(* Schneider Machine Expert - Basic project DFS, file version 2.5.0.0 *)
(* ProjectInformations: Name=New project *)

HARDWARE
  Cpu 0: TM221CE24R
  EthernetConfiguration: NetworkName=M221, IpAllocationMode=FixedAddress, IpAddress=0.0.0.0, SubnetMask=0.0.0.0
  SerialLineConfiguration: Baud=Baud19200, Parity=ParityEven, DataBits=DataBits8, StopBits=StopBits1, PhysicalMedium=PhysicalMediumRs485, TransmissionMode=TransmissionModeModbusRtu, SlaveId=1, Addressing=SlaveAddressing
  MastTask: UsePeriodScanMode=false, PeriodScan=100
  FastTask: Period=255
  CpuBehavior: StartingMode=StartAsPreviousState, AutoSaveRamOnEeprom=true, WatchdogPeriod=250

SYMBOLS  (address, symbol, comment, settings)
  %M0       SENSOR_JARAK_BIT
  %M1       LEVEL_BIT
  %M2       SM_BIT
  %M3       SB_BIT
  %M4       MOTOR_BIT
  %M5       WADAH_KT_BIT
  %M6       WADAH_KA_BIT
  %M7       MOTOR_TRIG
  %M8       KA_TRIGG
  %M9       KT_TRIG
  %I0.0     SENSOR_JARAK
  %I0.1     LEVEL
  %I0.2     SENSOR_MERAH
  %I0.3     SENSOR_BIRU
  %Q0.0     MOTOR_CONVEYOR
  %Q0.1     WADAH_KT
  %Q0.2     WADAH_KA

POU IO
  (* SectionNumber=0 *)

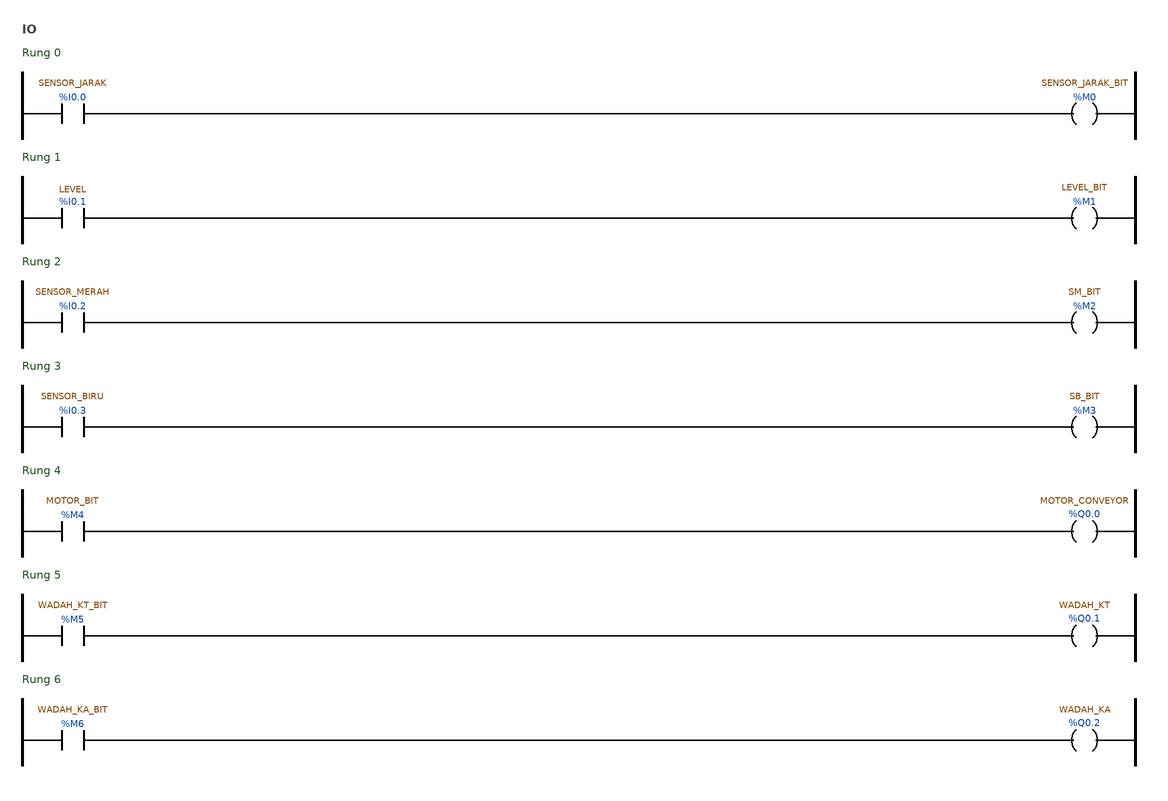

// Rung 0
  LD %I0.0                (* SENSOR_JARAK *)
  ST %M0                  (* SENSOR_JARAK_BIT *)
  // as ST:
  //   SENSOR_JARAK_BIT := SENSOR_JARAK;

// Rung 1
  LD %I0.1                (* LEVEL *)
  ST %M1                  (* LEVEL_BIT *)
  // as ST:
  //   LEVEL_BIT := LEVEL;

// Rung 2
  LD %I0.2                (* SENSOR_MERAH *)
  ST %M2                  (* SM_BIT *)
  // as ST:
  //   SM_BIT := SENSOR_MERAH;

// Rung 3
  LD %I0.3                (* SENSOR_BIRU *)
  ST %M3                  (* SB_BIT *)
  // as ST:
  //   SB_BIT := SENSOR_BIRU;

// Rung 4
  LD %M4                  (* MOTOR_BIT *)
  ST %Q0.0                (* MOTOR_CONVEYOR *)
  // as ST:
  //   MOTOR_CONVEYOR := MOTOR_BIT;

// Rung 5
  LD %M5                  (* WADAH_KT_BIT *)
  ST %Q0.1                (* WADAH_KT *)
  // as ST:
  //   WADAH_KT := WADAH_KT_BIT;

// Rung 6
  LD %M6                  (* WADAH_KA_BIT *)
  ST %Q0.2                (* WADAH_KA *)
  // as ST:
  //   WADAH_KA := WADAH_KA_BIT;

POU CONTROL
  (* SectionNumber=0 *)

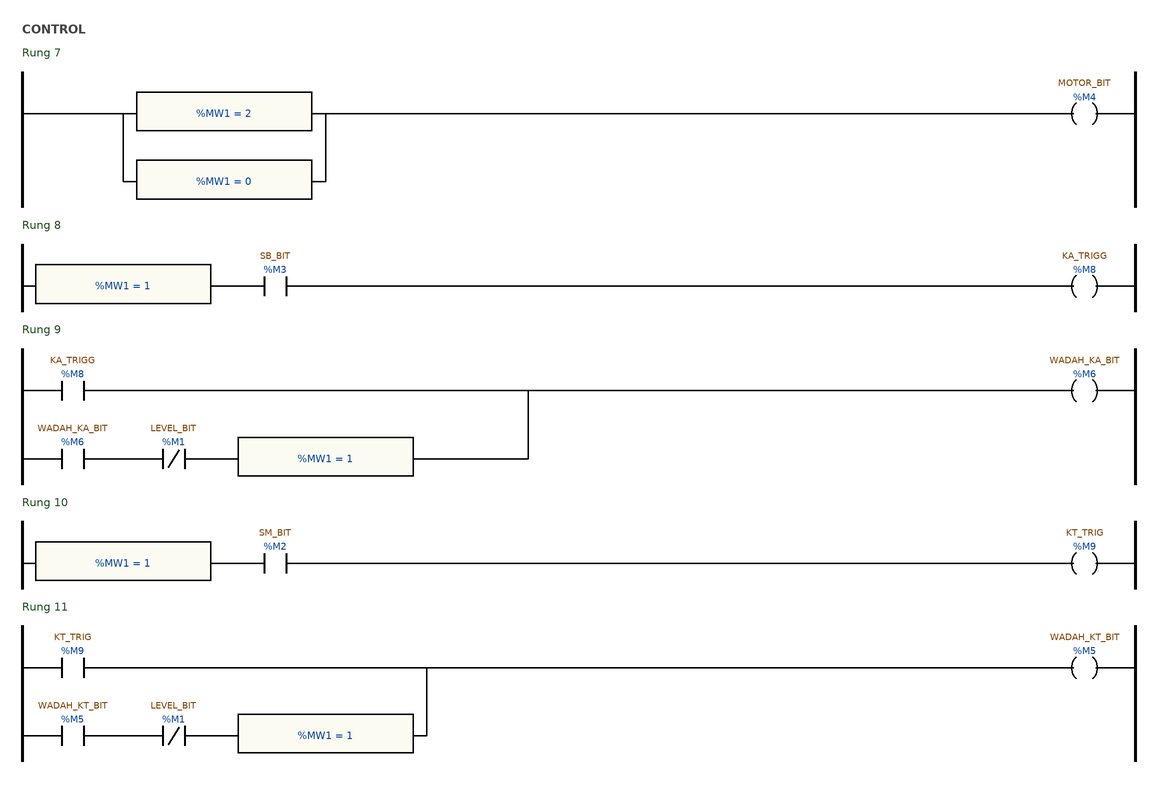

// Rung 7
  LD 1
  AND( [ %MW1 = 2 ]
  OR [ %MW1 = 0 ]
  )
  ST %M4                  (* MOTOR_BIT *)
  // as ST:
  //   MOTOR_BIT := %MW1 = 2 OR %MW1 = 0;

// Rung 8
  LD [ %MW1 = 1 ]
  AND %M3                 (* SB_BIT *)
  ST %M8                  (* KA_TRIGG *)
  // as ST:
  //   KA_TRIGG := %MW1 = 1 AND SB_BIT;

// Rung 9
  LD %M8                  (* KA_TRIGG *)
  OR( %M6                 (* WADAH_KA_BIT *)
  ANDN %M1                (* LEVEL_BIT *)
  AND [ %MW1 = 1 ]
  )
  ST %M6                  (* WADAH_KA_BIT *)
  // as ST:
  //   WADAH_KA_BIT := KA_TRIGG OR WADAH_KA_BIT AND NOT LEVEL_BIT AND %MW1 = 1;

// Rung 10
  LD [ %MW1 = 1 ]
  AND %M2                 (* SM_BIT *)
  ST %M9                  (* KT_TRIG *)
  // as ST:
  //   KT_TRIG := %MW1 = 1 AND SM_BIT;

// Rung 11
  LD %M9                  (* KT_TRIG *)
  OR( %M5                 (* WADAH_KT_BIT *)
  ANDN %M1                (* LEVEL_BIT *)
  AND [ %MW1 = 1 ]
  )
  ST %M5                  (* WADAH_KT_BIT *)
  // as ST:
  //   WADAH_KT_BIT := KT_TRIG OR WADAH_KT_BIT AND NOT LEVEL_BIT AND %MW1 = 1;

POU Siklus
  (* SectionNumber=0 *)

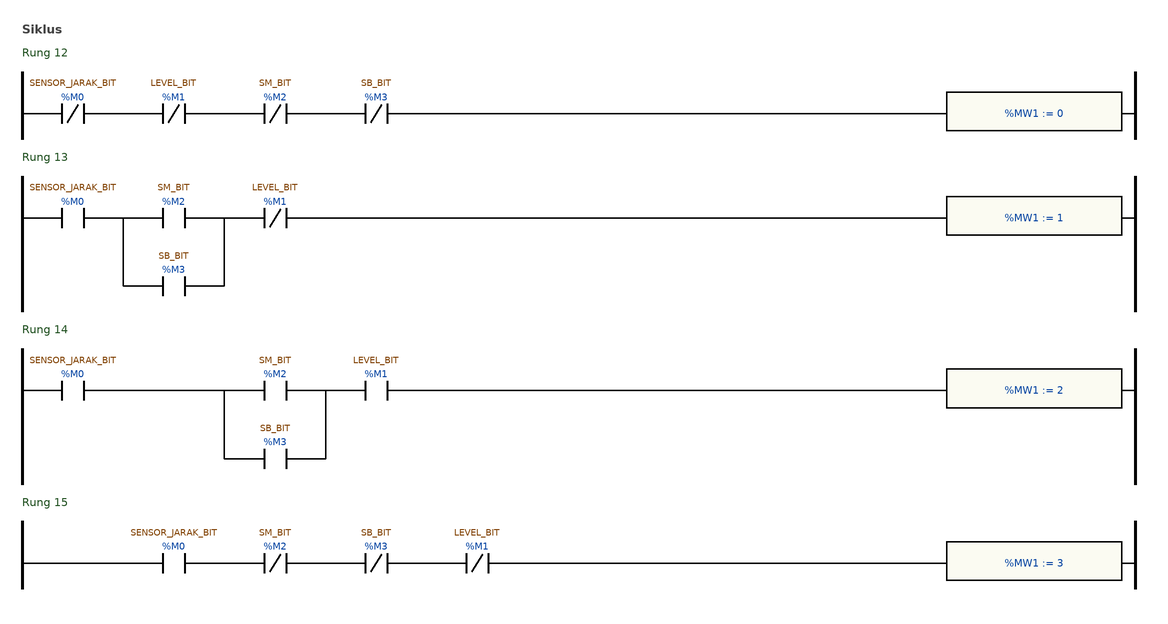

// Rung 12
  LDN %M0                 (* SENSOR_JARAK_BIT *)
  ANDN %M1                (* LEVEL_BIT *)
  ANDN %M2                (* SM_BIT *)
  ANDN %M3                (* SB_BIT *)
  [ %MW1 := 0 ]
  // as ST:
  //   IF NOT SENSOR_JARAK_BIT AND NOT LEVEL_BIT AND NOT SM_BIT AND NOT SB_BIT THEN %MW1 := 0; END_IF;

// Rung 13
  LD %M0                  (* SENSOR_JARAK_BIT *)
  AND( %M2                (* SM_BIT *)
  OR %M3                  (* SB_BIT *)
  )
  ANDN %M1                (* LEVEL_BIT *)
  [ %MW1 := 1 ]
  // as ST:
  //   IF SENSOR_JARAK_BIT AND (SM_BIT OR SB_BIT) AND NOT LEVEL_BIT THEN %MW1 := 1; END_IF;

// Rung 14
  LD %M0                  (* SENSOR_JARAK_BIT *)
  AND( %M2                (* SM_BIT *)
  OR %M3                  (* SB_BIT *)
  )
  AND %M1                 (* LEVEL_BIT *)
  [ %MW1 := 2 ]
  // as ST:
  //   IF SENSOR_JARAK_BIT AND (SM_BIT OR SB_BIT) AND LEVEL_BIT THEN %MW1 := 2; END_IF;

// Rung 15
  LD %M0                  (* SENSOR_JARAK_BIT *)
  ANDN %M2                (* SM_BIT *)
  ANDN %M3                (* SB_BIT *)
  ANDN %M1                (* LEVEL_BIT *)
  [ %MW1 := 3 ]
  // as ST:
  //   IF SENSOR_JARAK_BIT AND NOT SM_BIT AND NOT SB_BIT AND NOT LEVEL_BIT THEN %MW1 := 3; END_IF;
